FUNCTION GetArm3RotationPerpendicularToGround : LREAL
VAR_INPUT
	arm1RotationDegrees : LREAL;
	arm2RotationDegrees : LREAL;
END_VAR
VAR
END_VAR

GetArm3RotationPerpendicularToGround := -1.0 * (arm1RotationDegrees + arm2RotationDegrees);

END_FUNCTION

(* stored: Version 1.1.0.1, ProductVersion 3.1.4024.12
   POU GetArm3RotationPerpendicularToGround: Id {79deac1a-d420-49be-93ba-617f9889f39b}, SpecialFunc None *)
